FUNCTION_BLOCK RandomAddSupplier (* Composite Function Block Type *)
  (* Standard: 61499-2 *)
  (* Version 0.0, 11/21/2016, chivdan, nxtControl GmbH, template *)
  PACKAGE Main;
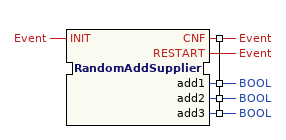
  EVENT_INPUT
    INIT; (* Initialization Request *)
  END_EVENT
  EVENT_OUTPUT
    CNF WITH add1, add2, add3; (* Initialization Confirm *)
    RESTART;
  END_EVENT
  VAR_OUTPUT
    add1 : BOOL;
    add2 : BOOL;
    add3 : BOOL;
  END_VAR
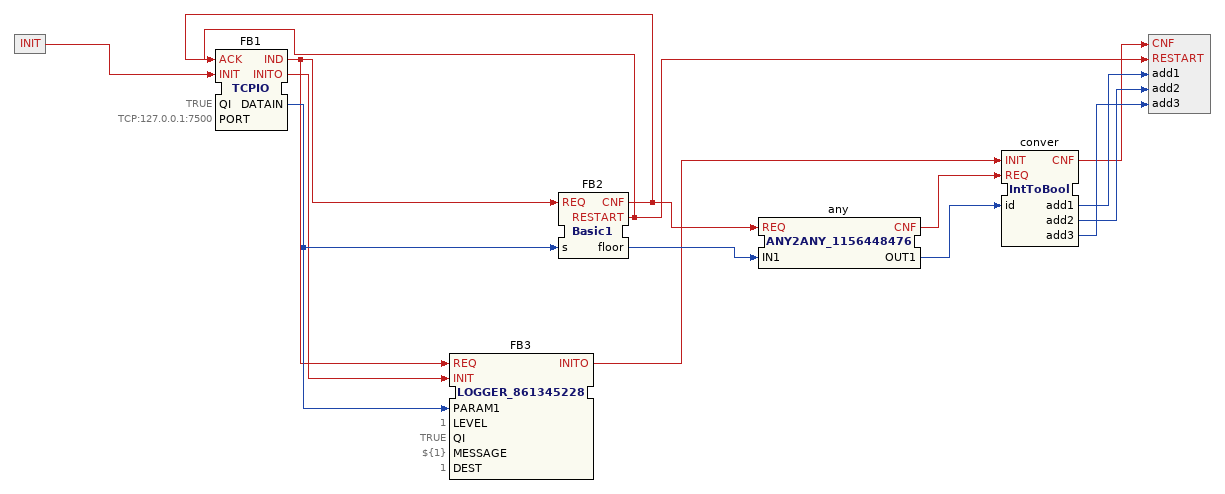
  FBS
    conver : IntToBool;
    any : ANY2ANY_1156448476; {SET_ATTRIBUTE(Configuration.GenericFBType.InterfaceParams, Runtime.Standard#CNT:=1;IN${CNT$}:STRING;OUT${CNT$}:INT)}
    FB1 : TCPIO(QI := TRUE, PORT := TCP:127.0.0.1:7500);
    FB2 : Basic1;
    FB3 : LOGGER_861345228(LEVEL := 1, QI := TRUE, MESSAGE := ${1}, DEST := 1); {SET_ATTRIBUTE(Configuration.GenericFBType.InterfaceParams, Runtime.System#CNT:=1)}
  END_FBS
  EVENT_CONNECTIONS
    any.CNF TO conver.REQ;
    FB1.IND TO FB2.REQ;
    FB2.CNF TO any.REQ;
    FB1.IND TO FB3.REQ;
    FB2.RESTART TO RESTART;
    FB2.CNF TO FB1.ACK;
    FB2.RESTART TO FB1.ACK;
    INIT TO FB1.INIT;
    FB1.INITO TO FB3.INIT;
    FB3.INITO TO conver.INIT;
    conver.CNF TO CNF;
  END_CONNECTIONS
  DATA_CONNECTIONS
    any.OUT1 TO conver.id;
    FB1.DATAIN TO FB2.s;
    FB2.floor TO any.IN1;
    FB1.DATAIN TO FB3.PARAM1;
    conver.add1 TO add1;
    conver.add2 TO add2;
    conver.add3 TO add3;
  END_CONNECTIONS
END_FUNCTION_BLOCK
